FUNCTION_BLOCK Desidratacao_HMI (* Service Interface Function Block Type *)
  (* Standard: 61499-2 *)
  (* Version 0.2, 11/05/2026, Faceplate Desidratacao. Comandos para cPressControl (cmdStsAutomatico, cmdHabilitaRevezamento, stpTempoRevezamentoCP1/2/3), CPress1/2/3 (cmdLigaCiclo + cmdResetFalha individuais), Preparador_Polimero1 (acmAutomatico, stsAutomatico). Display: almSemBombaDisp_1/2/3 + stsTempoRestante (sec/min/hora). DESIGN: status detalhado de M1..M5/VS1/FS1/ZSAH1/ZSAH2/Floculador de cada CPress eh exibido na faceplate INDIVIDUAL do CPress (publicado direto via SYMLINKMULTIVARSRC interno do bloco CPress). Mesmo design para Preparador_Polimero (faceplate propria). Reset global cmdResetFalhas: vai para BO/BR direto; supervisorio pulsa cmdResetFalha_CP1/2/3 individualmente para cobrir CPress. *)
  PACKAGE Hidryco.HidrycoLib;
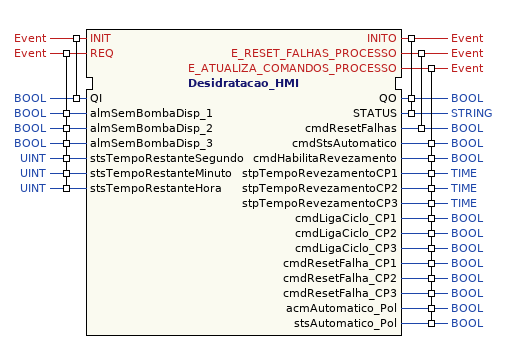
  EVENT_INPUT
    INIT WITH QI;
    REQ WITH almSemBombaDisp_1, almSemBombaDisp_2, almSemBombaDisp_3, stsTempoRestanteSegundo, stsTempoRestanteMinuto, stsTempoRestanteHora;
  END_EVENT
  EVENT_OUTPUT
    INITO WITH QO, STATUS;
    E_RESET_FALHAS_PROCESSO WITH cmdResetFalhas;
    E_ATUALIZA_COMANDOS_PROCESSO WITH cmdStsAutomatico, cmdHabilitaRevezamento, stpTempoRevezamentoCP1, stpTempoRevezamentoCP2, stpTempoRevezamentoCP3, cmdLigaCiclo_CP1, cmdLigaCiclo_CP2, cmdLigaCiclo_CP3, cmdResetFalha_CP1, cmdResetFalha_CP2, cmdResetFalha_CP3, acmAutomatico_Pol, stsAutomatico_Pol;
  END_EVENT
  VAR_INPUT
    QI : BOOL;
    almSemBombaDisp_1 : BOOL; (* Alarme: nenhuma bomba disponivel para C-Press 1 *)
    almSemBombaDisp_2 : BOOL; (* Alarme: nenhuma bomba disponivel para C-Press 2 *)
    almSemBombaDisp_3 : BOOL; (* Alarme: nenhuma bomba disponivel para C-Press 3 *)
    stsTempoRestanteSegundo : UINT; (* Tempo restante para revezamento (segundos) *)
    stsTempoRestanteMinuto : UINT; (* Tempo restante para revezamento (minutos) *)
    stsTempoRestanteHora : UINT; (* Tempo restante para revezamento (horas) *)
  END_VAR
  VAR_OUTPUT
    QO : BOOL; (* Event Output Qualifier *)
    STATUS : STRING; (* Service Status *)
    cmdResetFalhas : BOOL; (* Comando global de reset de falhas *)
    cmdStsAutomatico : BOOL; (* Operacao em automatico (cPressControl) *)
    cmdHabilitaRevezamento : BOOL; (* Habilita revezamento entre bombas de alimentacao *)
    stpTempoRevezamentoCP1 : TIME; (* Tempo de revezamento bomba BO_900_01 *)
    stpTempoRevezamentoCP2 : TIME; (* Tempo de revezamento bomba BO_900_02 *)
    stpTempoRevezamentoCP3 : TIME; (* Tempo de revezamento bomba BO_900_03 *)
    cmdLigaCiclo_CP1 : BOOL; (* Liga/Desliga ciclo CPress 1 (remoto) *)
    cmdLigaCiclo_CP2 : BOOL; (* Liga/Desliga ciclo CPress 2 (remoto) *)
    cmdLigaCiclo_CP3 : BOOL; (* Liga/Desliga ciclo CPress 3 (remoto) *)
    cmdResetFalha_CP1 : BOOL; (* Reset de falha CPress 1 *)
    cmdResetFalha_CP2 : BOOL; (* Reset de falha CPress 2 *)
    cmdResetFalha_CP3 : BOOL; (* Reset de falha CPress 3 *)
    acmAutomatico_Pol : BOOL; (* Acionamento automatico do Preparador de Polimero *)
    stsAutomatico_Pol : BOOL; (* Status automatico do Preparador de Polimero *)
  END_VAR
  SERVICE /
    SEQUENCE 
    END_SEQUENCE
  END_SERVICE
END_FUNCTION_BLOCK
